// TIA Portal V20 export
DATA_BLOCK "iDB_Conveyor_C2"   // DB413
// stored: Access Published, InstanceOfName Conveyor2.Conveyor_C2, InstanceOfType FB, Namespace Conveyor2
"Conveyor2.Conveyor_C2"
   // VAR
   //    Jog_Right : Bool;
   //    Jog_Left : Bool;
   //    Auto_Right : Bool;
   //    PF_Bay1_NewProd : Bool;
   //    PF_Bay2_NewProd : Bool;
   //    PF_Bay3_NewProd : Bool;
   //    PF_Bay4_EndConv : Bool;
   // END_VAR
BEGIN
END_DATA_BLOCK
